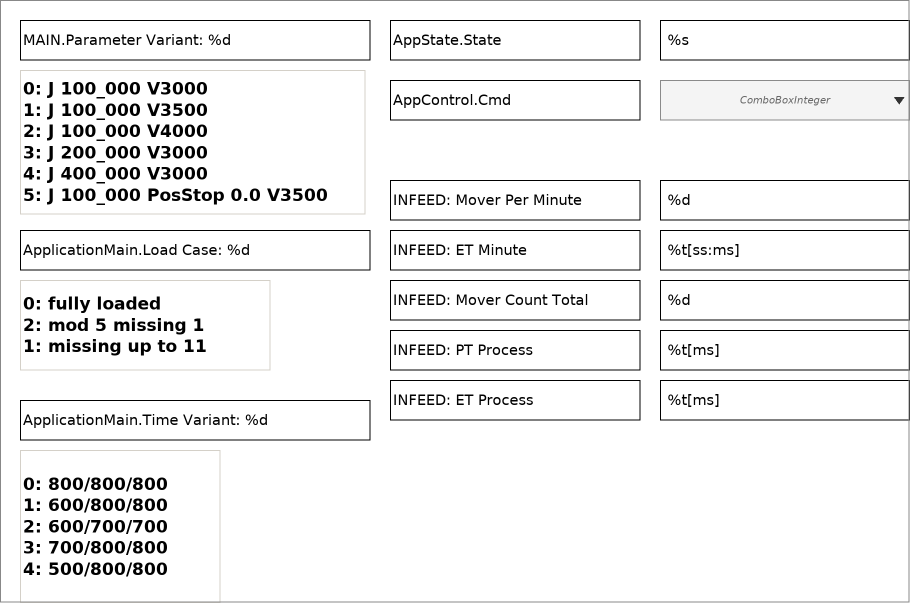
VISUALIZATION SIM_TEST  // 910x603
    Rectangle (20,230 350x40), "ApplicationMain.Load Case: %d", text variable: GVL_APPLICATION.ApplicationMain._nLoadCase
        OnMouseClick: write the text variable via VisuDialogs.Numpad, min 0, max 2
    Rectangle (20,400 350x40), "ApplicationMain.Time Variant: %d", text variable: GVL_APPLICATION.ApplicationMain._nTimeVariant
        OnMouseClick: write the text variable via VisuDialogs.Numpad, min 0, max 100
    Rectangle (20,20 350x40), "MAIN.Parameter Variant: %d", text variable: MAIN.nParameterVariant
        toggle MAIN.bWriteVariant
        OnMouseClick: write the text variable via VisuDialogs.Numpad, min 0, max 100
    Textfield (20,450 200x153), "0: 800/800/800 1: 600/800/800 2: 600/700/700 3: 700/800/800 4: 500/800/800"
    Textfield (20,280 250x90), "0: fully loaded 2: mod 5 missing 1 1: missing up to 11"
    Textfield (20,70 345x144), "0: J 100_000 V3000 1: J 100_000 V3500 2: J 100_000 V4000 3: J 200_000 V3000 4: J 400_000 V3000 5: J 100_000 PosStop 0.0 V3500"
    Rectangle (390,80 250x40), "AppControl.Cmd"
    ComboBoxInteger (660,80 250x40), variable: GVL_APPLICATION.AppControl.Cmd, text list: 'TL_E_INSTANCE_CMD'
    Rectangle (390,20 250x40), "AppState.State"
    Rectangle (660,20 250x40), "%s", text variable: GVL_APPLICATION.ApplicationMain._sAppState
    Rectangle (390,180 250x40), "INFEED: Mover Per Minute"
    Rectangle (660,180 250x40), "%d", text variable: GVL_APPLICATION.ProcessCollector[2]._AllStationMoverPerMinute
    Rectangle (390,280 250x40), "INFEED: Mover Count Total"
    Rectangle (660,280 250x40), "%d", text variable: GVL_APPLICATION.ProcessCollector[2]._nMoverCountTotal
    Rectangle (390,380 250x40), "INFEED: ET Process"
    Rectangle (660,380 250x40), "%t[ms]", text variable: GVL_APPLICATION.ApplicationMain._tonProcess[2].ET
    Rectangle (390,330 250x40), "INFEED: PT Process"
    Rectangle (660,330 250x40), "%t[ms]", text variable: GVL_APPLICATION.ApplicationMain._tProcess[2]
    Rectangle (390,230 250x40), "INFEED: ET Minute"
    Rectangle (660,230 250x40), "%t[ss:ms]", text variable: ProcessCollector[2]._tonPartsPerMinute.ET
END_VISUALIZATION

(* stored: Version 1.1.0.1, ProductVersion 3.1.4026.12
   Visu SIM_TEST: Id {986ae958-2a9d-4eb4-9e8a-0f993c444b4f} *)
